(* PLC project linear_function, Dassault Systèmes ControlBuild 2024x *)
(* stored: creationDateTime 2023-10-03T11:13:30-01:00 *)

(* This module simulates the evolution of a ramp in function of a real input. The equation form is (y = ax + b). *)
FUNCTION_BLOCK equipment_library.linear_function
  VAR_INPUT
    input : REAL := 0.0;
  END_VAR
  VAR_OUTPUT
    output : REAL := 0.0;
  END_VAR
  VAR CONSTANT
    a : REAL := 1.0;
    b : REAL := 0.0;
  END_VAR


ACTION C_source_code:
/* ----------------------------------------------------------------	*/
/* Type : Model of Operative Behaviour					*/
/* Category :  Toolbox							*/
/* Author : Dassault Systemes						*/
/* Update date : June 2018						*/
/* ----------------------------------------------------------------	*/
/* This module simulates the evolution of a  ramp 			*/
/*	in function of a real input.					*/
/* The equation's form is y = ax + b.					*/
/* ----------------------------------------------------------------	*/

output =a*input + b;
END_ACTION
END_FUNCTION_BLOCK
